TYPE DeviceDataExt EXTENDS DeviceData :
STRUCT
	Justified: BOOL;
	ClingRequired: BOOL;
	ClingSize: cClingSize;
	CartonNum: DINT;
	CartonTracking: DINT;
	ToteRFID: DINT;
	ToteSide: DINT; //TODO, used for 1 or 2 phones in tote, to be removed
	JustifyNest: DINT;
END_STRUCT
END_TYPE

(* stored: Version 1.1.0.1, ProductVersion 3.1.4024.6
   DUT DeviceDataExt: Id {a70c4000-98e6-4ae5-b8e0-be7854b673b8} *)
